// TwinCAT 3 PLC project PLC1
// ProgramVersion: 3.1.4023.0
// libraries:
//   Tc2_Standard, * (Beckhoff Automation GmbH)
//   Tc2_System, * (Beckhoff Automation GmbH)
//   Tc3_Module, * (Beckhoff Automation GmbH)
// project tree:
//   / PlcTask.TcTTO
//   POUs/ MAIN.TcPOU
// real-time tasks:
//   TASK PlcTask: cycle T#10ms, priority 20, ADS port 350
// I/O:
//   DEVICE Device 1 (EtherCAT), AmsNetId 5.48.71.138.2.1
//     Term 1 (EK1200) [EK1200-5000 EtherCAT Power supply (2A E-Bus)]
//       Term 2 (EL1004) [EL1004 4Ch. Dig. Input 24V, 3ms]
//       Term 3 (EL2004) [EL2004 4Ch. Dig. Output 24V, 0.5A]
//       Term 4 (EL3102) [EL3102 2Ch. Ana. Input +/-10V, Diff.]
//       Term 5 (EL9011) [EL9011 End Terminal]
// variable links:
//   PLC1/PLC1 Instance <-> Device 1 (EtherCAT)/Term 1 (EK1200)/Term 2 (EL1004)
//     PlcTask Inputs/MAIN.bDin <-> Channel 1/Input
//   PLC1/PLC1 Instance <-> Device 1 (EtherCAT)/Term 1 (EK1200)/Term 4 (EL3102)
//     PlcTask Inputs/MAIN.nAin <-> AI Standard Channel 1/Value

CONFIGURATION PLC1
    RESOURCE PLC ON TwinCAT3
        TASK PlcTask(INTERVAL := T#10ms, PRIORITY := 20);
        PROGRAM MAIN WITH PlcTask : MAIN;
    END_RESOURCE
END_CONFIGURATION

// ---- POUs/MAIN.TcPOU
PROGRAM MAIN
VAR
	bDin AT %I*: BOOL;	
	nAin AT %I*: INT;
	
	nSin: LREAL;
	fbton: TON;
	nTemp: REAL;
	{attribute 'TcAnalytics'}
	bDinx: BOOL;
	{attribute 'TcAnalytics'}
	nAinx: INT;
END_VAR

fbton(IN:= NOT fbton.Q,PT:= T#100MS);
IF fbton.Q THEN
	nTemp:= nTemp + 0.1;
	IF nTemp >= 3.2 THEN
		nTemp := 0;
	END_IF
END_IF
nSin := 100*SIN(nTemp);
bDinx:= bDin;
nAinx:= nAin;

END_PROGRAM
